TYPE ST_Netcontactor_set :
STRUCT
	e_ACRotationState				: eACRotationState; // 0:No AC, 1: AC CLOCKWISE, 2: AC ANTI-CLOCKWISE
	e_ClosingRequest				: eNetcontMode;
	b_ACdetected					: BOOL;
	b_RotationSwitchEnable			: BOOL;
	b_SynchronizedToD7				: BOOL;
END_STRUCT
END_TYPE

(* stored: Version 1.1.0.1, ProductVersion 3.1.4026.18
   DUT ST_Netcontactor_set: Id {b4b69345-3296-4468-915c-4d0bb03897b5} *)
